TYPE fbPistonStatus :
STRUCT
	AtHome : TIME;
	AtWork : TIME;
END_STRUCT
END_TYPE

(* stored: Version 1.1.0.1, ProductVersion 3.1.4024.9
   DUT fbPistonStatus: Id {a2ab828e-f095-0ceb-1bea-12d13845e051} *)
